// TIA Portal V18 export
FUNCTION "HeatingPLC_vIO" : Void   // FC11001, LAD
{ S7_Optimized_Access := 'FALSE' }
VERSION : 0.1
// stored: AutoNumber false, IsIECCheckEnabled false, SetENOAutomatically false, UDAEnableTagReadback false
BEGIN

REGION Network 1
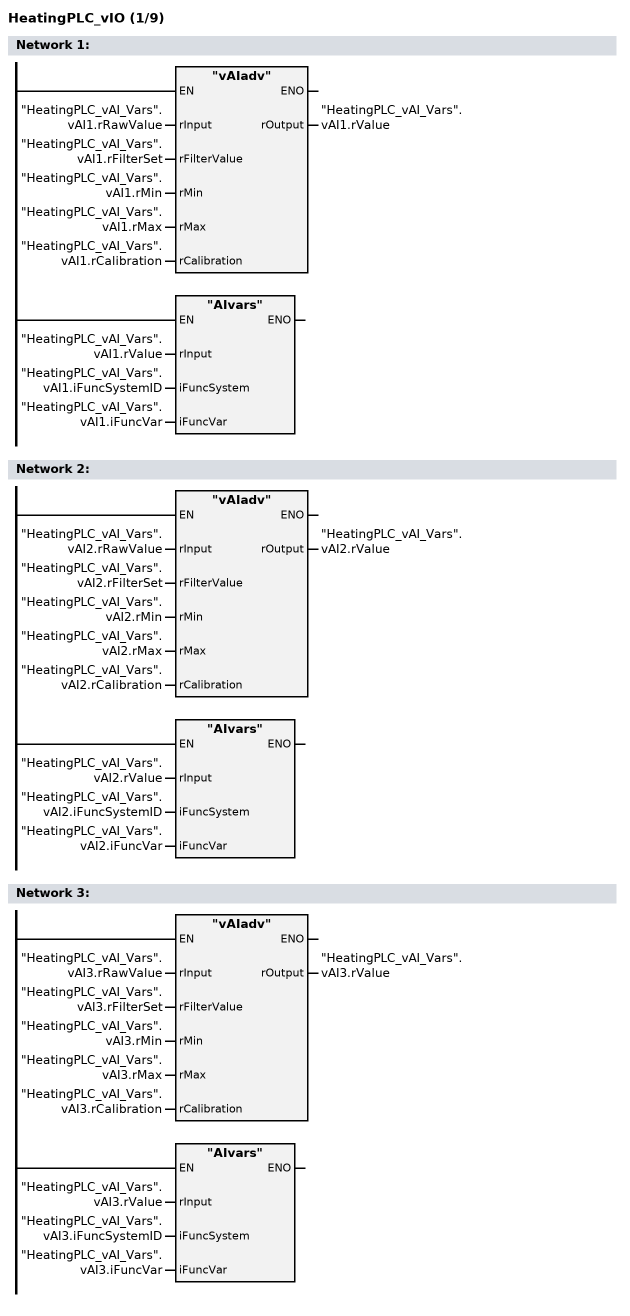
   RUNG wire#powerrail
      "vAIadv"(rInput := "HeatingPLC_vAI_Vars".vAI1.rRawValue, rFilterValue := "HeatingPLC_vAI_Vars".vAI1.rFilterSet, rMin := "HeatingPLC_vAI_Vars".vAI1.rMin, rMax := "HeatingPLC_vAI_Vars".vAI1.rMax, rCalibration := "HeatingPLC_vAI_Vars".vAI1.rCalibration, rOutput => "HeatingPLC_vAI_Vars".vAI1.rValue)
   END_RUNG
   RUNG wire#powerrail
      "AIvars"(rInput := "HeatingPLC_vAI_Vars".vAI1.rValue, iFuncSystem := "HeatingPLC_vAI_Vars".vAI1.iFuncSystemID, iFuncVar := "HeatingPLC_vAI_Vars".vAI1.iFuncVar)
   END_RUNG
   // the same network as SCL:
   "vAIadv"(rInput := "HeatingPLC_vAI_Vars".vAI1.rRawValue,
            rFilterValue := "HeatingPLC_vAI_Vars".vAI1.rFilterSet,
            rMin := "HeatingPLC_vAI_Vars".vAI1.rMin,
            rMax := "HeatingPLC_vAI_Vars".vAI1.rMax,
            rCalibration := "HeatingPLC_vAI_Vars".vAI1.rCalibration,
            rOutput => "HeatingPLC_vAI_Vars".vAI1.rValue);
   "AIvars"(rInput := "HeatingPLC_vAI_Vars".vAI1.rValue,
            iFuncSystem := "HeatingPLC_vAI_Vars".vAI1.iFuncSystemID,
            iFuncVar := "HeatingPLC_vAI_Vars".vAI1.iFuncVar);
END_REGION

REGION Network 2
   RUNG wire#powerrail
      "vAIadv"(rInput := "HeatingPLC_vAI_Vars".vAI2.rRawValue, rFilterValue := "HeatingPLC_vAI_Vars".vAI2.rFilterSet, rMin := "HeatingPLC_vAI_Vars".vAI2.rMin, rMax := "HeatingPLC_vAI_Vars".vAI2.rMax, rCalibration := "HeatingPLC_vAI_Vars".vAI2.rCalibration, rOutput => "HeatingPLC_vAI_Vars".vAI2.rValue)
   END_RUNG
   RUNG wire#powerrail
      "AIvars"(rInput := "HeatingPLC_vAI_Vars".vAI2.rValue, iFuncSystem := "HeatingPLC_vAI_Vars".vAI2.iFuncSystemID, iFuncVar := "HeatingPLC_vAI_Vars".vAI2.iFuncVar)
   END_RUNG
   // the same network as SCL:
   "vAIadv"(rInput := "HeatingPLC_vAI_Vars".vAI2.rRawValue,
            rFilterValue := "HeatingPLC_vAI_Vars".vAI2.rFilterSet,
            rMin := "HeatingPLC_vAI_Vars".vAI2.rMin,
            rMax := "HeatingPLC_vAI_Vars".vAI2.rMax,
            rCalibration := "HeatingPLC_vAI_Vars".vAI2.rCalibration,
            rOutput => "HeatingPLC_vAI_Vars".vAI2.rValue);
   "AIvars"(rInput := "HeatingPLC_vAI_Vars".vAI2.rValue,
            iFuncSystem := "HeatingPLC_vAI_Vars".vAI2.iFuncSystemID,
            iFuncVar := "HeatingPLC_vAI_Vars".vAI2.iFuncVar);
END_REGION

REGION Network 3
   RUNG wire#powerrail
      "vAIadv"(rInput := "HeatingPLC_vAI_Vars".vAI3.rRawValue, rFilterValue := "HeatingPLC_vAI_Vars".vAI3.rFilterSet, rMin := "HeatingPLC_vAI_Vars".vAI3.rMin, rMax := "HeatingPLC_vAI_Vars".vAI3.rMax, rCalibration := "HeatingPLC_vAI_Vars".vAI3.rCalibration, rOutput => "HeatingPLC_vAI_Vars".vAI3.rValue)
   END_RUNG
   RUNG wire#powerrail
      "AIvars"(rInput := "HeatingPLC_vAI_Vars".vAI3.rValue, iFuncSystem := "HeatingPLC_vAI_Vars".vAI3.iFuncSystemID, iFuncVar := "HeatingPLC_vAI_Vars".vAI3.iFuncVar)
   END_RUNG
   // the same network as SCL:
   "vAIadv"(rInput := "HeatingPLC_vAI_Vars".vAI3.rRawValue,
            rFilterValue := "HeatingPLC_vAI_Vars".vAI3.rFilterSet,
            rMin := "HeatingPLC_vAI_Vars".vAI3.rMin,
            rMax := "HeatingPLC_vAI_Vars".vAI3.rMax,
            rCalibration := "HeatingPLC_vAI_Vars".vAI3.rCalibration,
            rOutput => "HeatingPLC_vAI_Vars".vAI3.rValue);
   "AIvars"(rInput := "HeatingPLC_vAI_Vars".vAI3.rValue,
            iFuncSystem := "HeatingPLC_vAI_Vars".vAI3.iFuncSystemID,
            iFuncVar := "HeatingPLC_vAI_Vars".vAI3.iFuncVar);
END_REGION

REGION Network 4
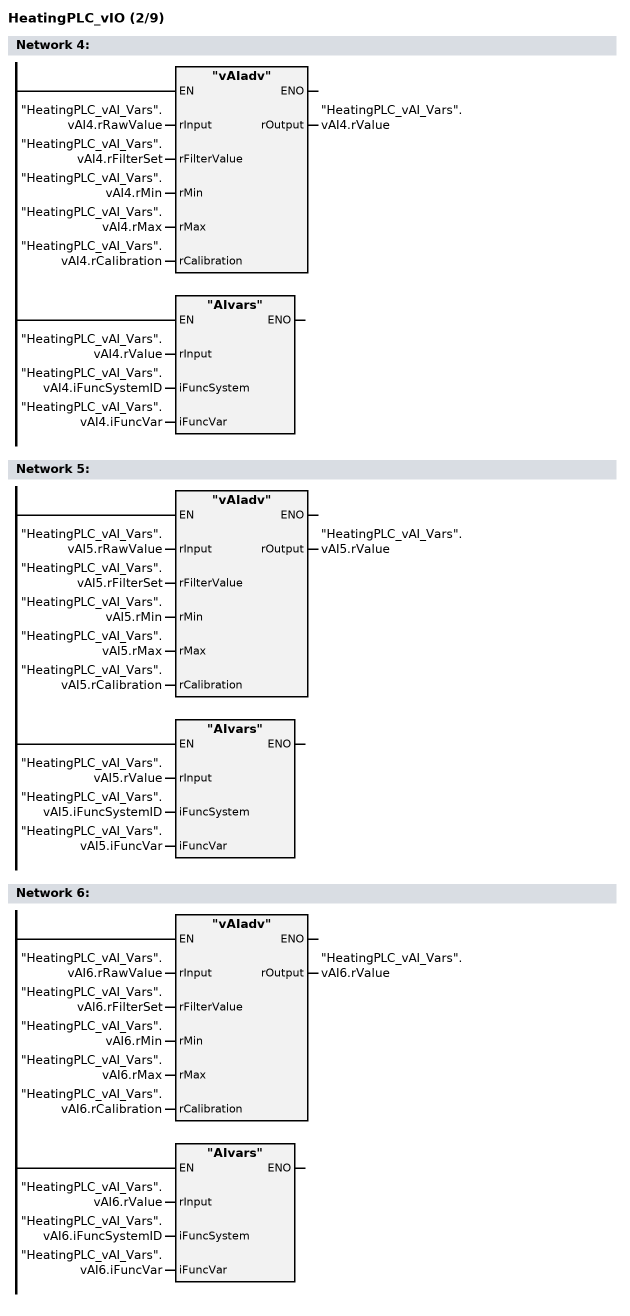
   RUNG wire#powerrail
      "vAIadv"(rInput := "HeatingPLC_vAI_Vars".vAI4.rRawValue, rFilterValue := "HeatingPLC_vAI_Vars".vAI4.rFilterSet, rMin := "HeatingPLC_vAI_Vars".vAI4.rMin, rMax := "HeatingPLC_vAI_Vars".vAI4.rMax, rCalibration := "HeatingPLC_vAI_Vars".vAI4.rCalibration, rOutput => "HeatingPLC_vAI_Vars".vAI4.rValue)
   END_RUNG
   RUNG wire#powerrail
      "AIvars"(rInput := "HeatingPLC_vAI_Vars".vAI4.rValue, iFuncSystem := "HeatingPLC_vAI_Vars".vAI4.iFuncSystemID, iFuncVar := "HeatingPLC_vAI_Vars".vAI4.iFuncVar)
   END_RUNG
   // the same network as SCL:
   "vAIadv"(rInput := "HeatingPLC_vAI_Vars".vAI4.rRawValue,
            rFilterValue := "HeatingPLC_vAI_Vars".vAI4.rFilterSet,
            rMin := "HeatingPLC_vAI_Vars".vAI4.rMin,
            rMax := "HeatingPLC_vAI_Vars".vAI4.rMax,
            rCalibration := "HeatingPLC_vAI_Vars".vAI4.rCalibration,
            rOutput => "HeatingPLC_vAI_Vars".vAI4.rValue);
   "AIvars"(rInput := "HeatingPLC_vAI_Vars".vAI4.rValue,
            iFuncSystem := "HeatingPLC_vAI_Vars".vAI4.iFuncSystemID,
            iFuncVar := "HeatingPLC_vAI_Vars".vAI4.iFuncVar);
END_REGION

REGION Network 5
   RUNG wire#powerrail
      "vAIadv"(rInput := "HeatingPLC_vAI_Vars".vAI5.rRawValue, rFilterValue := "HeatingPLC_vAI_Vars".vAI5.rFilterSet, rMin := "HeatingPLC_vAI_Vars".vAI5.rMin, rMax := "HeatingPLC_vAI_Vars".vAI5.rMax, rCalibration := "HeatingPLC_vAI_Vars".vAI5.rCalibration, rOutput => "HeatingPLC_vAI_Vars".vAI5.rValue)
   END_RUNG
   RUNG wire#powerrail
      "AIvars"(rInput := "HeatingPLC_vAI_Vars".vAI5.rValue, iFuncSystem := "HeatingPLC_vAI_Vars".vAI5.iFuncSystemID, iFuncVar := "HeatingPLC_vAI_Vars".vAI5.iFuncVar)
   END_RUNG
   // the same network as SCL:
   "vAIadv"(rInput := "HeatingPLC_vAI_Vars".vAI5.rRawValue,
            rFilterValue := "HeatingPLC_vAI_Vars".vAI5.rFilterSet,
            rMin := "HeatingPLC_vAI_Vars".vAI5.rMin,
            rMax := "HeatingPLC_vAI_Vars".vAI5.rMax,
            rCalibration := "HeatingPLC_vAI_Vars".vAI5.rCalibration,
            rOutput => "HeatingPLC_vAI_Vars".vAI5.rValue);
   "AIvars"(rInput := "HeatingPLC_vAI_Vars".vAI5.rValue,
            iFuncSystem := "HeatingPLC_vAI_Vars".vAI5.iFuncSystemID,
            iFuncVar := "HeatingPLC_vAI_Vars".vAI5.iFuncVar);
END_REGION

REGION Network 6
   RUNG wire#powerrail
      "vAIadv"(rInput := "HeatingPLC_vAI_Vars".vAI6.rRawValue, rFilterValue := "HeatingPLC_vAI_Vars".vAI6.rFilterSet, rMin := "HeatingPLC_vAI_Vars".vAI6.rMin, rMax := "HeatingPLC_vAI_Vars".vAI6.rMax, rCalibration := "HeatingPLC_vAI_Vars".vAI6.rCalibration, rOutput => "HeatingPLC_vAI_Vars".vAI6.rValue)
   END_RUNG
   RUNG wire#powerrail
      "AIvars"(rInput := "HeatingPLC_vAI_Vars".vAI6.rValue, iFuncSystem := "HeatingPLC_vAI_Vars".vAI6.iFuncSystemID, iFuncVar := "HeatingPLC_vAI_Vars".vAI6.iFuncVar)
   END_RUNG
   // the same network as SCL:
   "vAIadv"(rInput := "HeatingPLC_vAI_Vars".vAI6.rRawValue,
            rFilterValue := "HeatingPLC_vAI_Vars".vAI6.rFilterSet,
            rMin := "HeatingPLC_vAI_Vars".vAI6.rMin,
            rMax := "HeatingPLC_vAI_Vars".vAI6.rMax,
            rCalibration := "HeatingPLC_vAI_Vars".vAI6.rCalibration,
            rOutput => "HeatingPLC_vAI_Vars".vAI6.rValue);
   "AIvars"(rInput := "HeatingPLC_vAI_Vars".vAI6.rValue,
            iFuncSystem := "HeatingPLC_vAI_Vars".vAI6.iFuncSystemID,
            iFuncVar := "HeatingPLC_vAI_Vars".vAI6.iFuncVar);
END_REGION

REGION Network 7
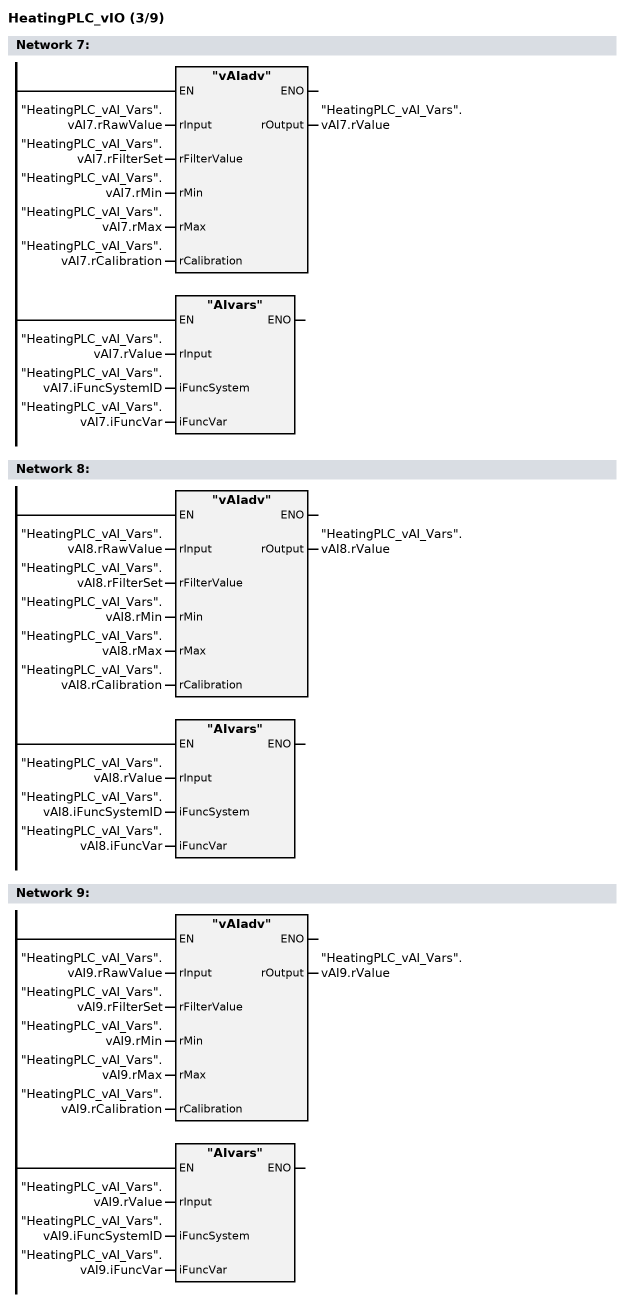
   RUNG wire#powerrail
      "vAIadv"(rInput := "HeatingPLC_vAI_Vars".vAI7.rRawValue, rFilterValue := "HeatingPLC_vAI_Vars".vAI7.rFilterSet, rMin := "HeatingPLC_vAI_Vars".vAI7.rMin, rMax := "HeatingPLC_vAI_Vars".vAI7.rMax, rCalibration := "HeatingPLC_vAI_Vars".vAI7.rCalibration, rOutput => "HeatingPLC_vAI_Vars".vAI7.rValue)
   END_RUNG
   RUNG wire#powerrail
      "AIvars"(rInput := "HeatingPLC_vAI_Vars".vAI7.rValue, iFuncSystem := "HeatingPLC_vAI_Vars".vAI7.iFuncSystemID, iFuncVar := "HeatingPLC_vAI_Vars".vAI7.iFuncVar)
   END_RUNG
   // the same network as SCL:
   "vAIadv"(rInput := "HeatingPLC_vAI_Vars".vAI7.rRawValue,
            rFilterValue := "HeatingPLC_vAI_Vars".vAI7.rFilterSet,
            rMin := "HeatingPLC_vAI_Vars".vAI7.rMin,
            rMax := "HeatingPLC_vAI_Vars".vAI7.rMax,
            rCalibration := "HeatingPLC_vAI_Vars".vAI7.rCalibration,
            rOutput => "HeatingPLC_vAI_Vars".vAI7.rValue);
   "AIvars"(rInput := "HeatingPLC_vAI_Vars".vAI7.rValue,
            iFuncSystem := "HeatingPLC_vAI_Vars".vAI7.iFuncSystemID,
            iFuncVar := "HeatingPLC_vAI_Vars".vAI7.iFuncVar);
END_REGION

REGION Network 8
   RUNG wire#powerrail
      "vAIadv"(rInput := "HeatingPLC_vAI_Vars".vAI8.rRawValue, rFilterValue := "HeatingPLC_vAI_Vars".vAI8.rFilterSet, rMin := "HeatingPLC_vAI_Vars".vAI8.rMin, rMax := "HeatingPLC_vAI_Vars".vAI8.rMax, rCalibration := "HeatingPLC_vAI_Vars".vAI8.rCalibration, rOutput => "HeatingPLC_vAI_Vars".vAI8.rValue)
   END_RUNG
   RUNG wire#powerrail
      "AIvars"(rInput := "HeatingPLC_vAI_Vars".vAI8.rValue, iFuncSystem := "HeatingPLC_vAI_Vars".vAI8.iFuncSystemID, iFuncVar := "HeatingPLC_vAI_Vars".vAI8.iFuncVar)
   END_RUNG
   // the same network as SCL:
   "vAIadv"(rInput := "HeatingPLC_vAI_Vars".vAI8.rRawValue,
            rFilterValue := "HeatingPLC_vAI_Vars".vAI8.rFilterSet,
            rMin := "HeatingPLC_vAI_Vars".vAI8.rMin,
            rMax := "HeatingPLC_vAI_Vars".vAI8.rMax,
            rCalibration := "HeatingPLC_vAI_Vars".vAI8.rCalibration,
            rOutput => "HeatingPLC_vAI_Vars".vAI8.rValue);
   "AIvars"(rInput := "HeatingPLC_vAI_Vars".vAI8.rValue,
            iFuncSystem := "HeatingPLC_vAI_Vars".vAI8.iFuncSystemID,
            iFuncVar := "HeatingPLC_vAI_Vars".vAI8.iFuncVar);
END_REGION

REGION Network 9
   RUNG wire#powerrail
      "vAIadv"(rInput := "HeatingPLC_vAI_Vars".vAI9.rRawValue, rFilterValue := "HeatingPLC_vAI_Vars".vAI9.rFilterSet, rMin := "HeatingPLC_vAI_Vars".vAI9.rMin, rMax := "HeatingPLC_vAI_Vars".vAI9.rMax, rCalibration := "HeatingPLC_vAI_Vars".vAI9.rCalibration, rOutput => "HeatingPLC_vAI_Vars".vAI9.rValue)
   END_RUNG
   RUNG wire#powerrail
      "AIvars"(rInput := "HeatingPLC_vAI_Vars".vAI9.rValue, iFuncSystem := "HeatingPLC_vAI_Vars".vAI9.iFuncSystemID, iFuncVar := "HeatingPLC_vAI_Vars".vAI9.iFuncVar)
   END_RUNG
   // the same network as SCL:
   "vAIadv"(rInput := "HeatingPLC_vAI_Vars".vAI9.rRawValue,
            rFilterValue := "HeatingPLC_vAI_Vars".vAI9.rFilterSet,
            rMin := "HeatingPLC_vAI_Vars".vAI9.rMin,
            rMax := "HeatingPLC_vAI_Vars".vAI9.rMax,
            rCalibration := "HeatingPLC_vAI_Vars".vAI9.rCalibration,
            rOutput => "HeatingPLC_vAI_Vars".vAI9.rValue);
   "AIvars"(rInput := "HeatingPLC_vAI_Vars".vAI9.rValue,
            iFuncSystem := "HeatingPLC_vAI_Vars".vAI9.iFuncSystemID,
            iFuncVar := "HeatingPLC_vAI_Vars".vAI9.iFuncVar);
END_REGION

REGION Network 10
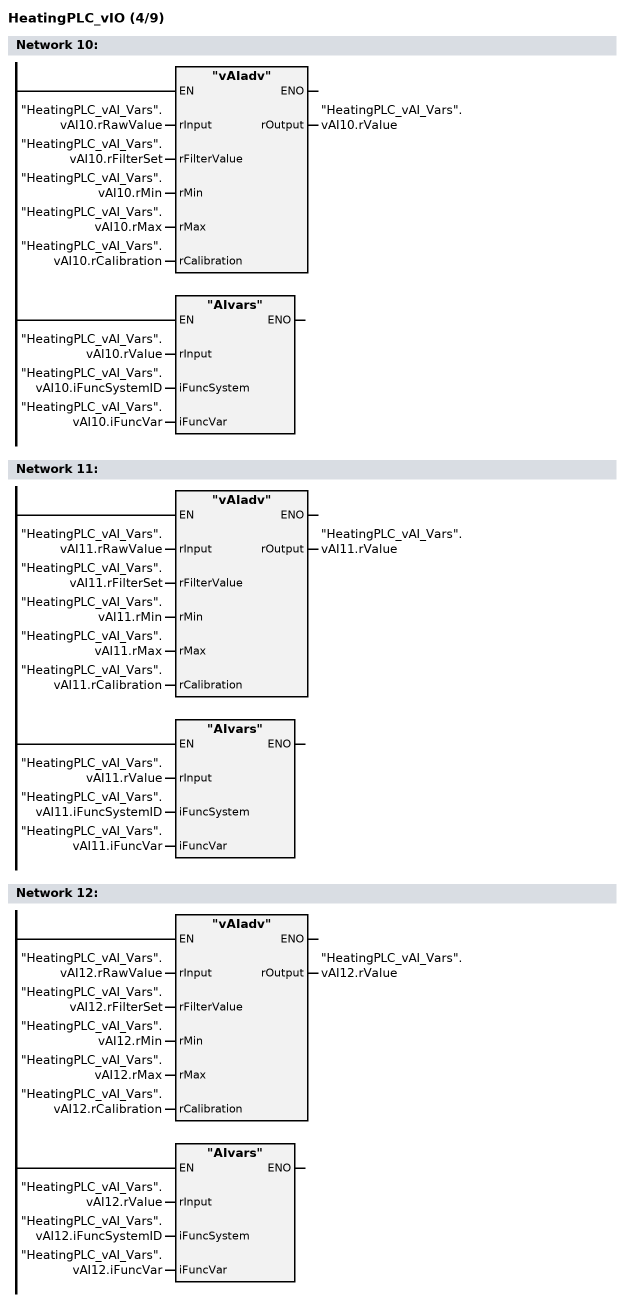
   RUNG wire#powerrail
      "vAIadv"(rInput := "HeatingPLC_vAI_Vars".vAI10.rRawValue, rFilterValue := "HeatingPLC_vAI_Vars".vAI10.rFilterSet, rMin := "HeatingPLC_vAI_Vars".vAI10.rMin, rMax := "HeatingPLC_vAI_Vars".vAI10.rMax, rCalibration := "HeatingPLC_vAI_Vars".vAI10.rCalibration, rOutput => "HeatingPLC_vAI_Vars".vAI10.rValue)
   END_RUNG
   RUNG wire#powerrail
      "AIvars"(rInput := "HeatingPLC_vAI_Vars".vAI10.rValue, iFuncSystem := "HeatingPLC_vAI_Vars".vAI10.iFuncSystemID, iFuncVar := "HeatingPLC_vAI_Vars".vAI10.iFuncVar)
   END_RUNG
   // the same network as SCL:
   "vAIadv"(rInput := "HeatingPLC_vAI_Vars".vAI10.rRawValue,
            rFilterValue := "HeatingPLC_vAI_Vars".vAI10.rFilterSet,
            rMin := "HeatingPLC_vAI_Vars".vAI10.rMin,
            rMax := "HeatingPLC_vAI_Vars".vAI10.rMax,
            rCalibration := "HeatingPLC_vAI_Vars".vAI10.rCalibration,
            rOutput => "HeatingPLC_vAI_Vars".vAI10.rValue);
   "AIvars"(rInput := "HeatingPLC_vAI_Vars".vAI10.rValue,
            iFuncSystem := "HeatingPLC_vAI_Vars".vAI10.iFuncSystemID,
            iFuncVar := "HeatingPLC_vAI_Vars".vAI10.iFuncVar);
END_REGION

REGION Network 11
   RUNG wire#powerrail
      "vAIadv"(rInput := "HeatingPLC_vAI_Vars".vAI11.rRawValue, rFilterValue := "HeatingPLC_vAI_Vars".vAI11.rFilterSet, rMin := "HeatingPLC_vAI_Vars".vAI11.rMin, rMax := "HeatingPLC_vAI_Vars".vAI11.rMax, rCalibration := "HeatingPLC_vAI_Vars".vAI11.rCalibration, rOutput => "HeatingPLC_vAI_Vars".vAI11.rValue)
   END_RUNG
   RUNG wire#powerrail
      "AIvars"(rInput := "HeatingPLC_vAI_Vars".vAI11.rValue, iFuncSystem := "HeatingPLC_vAI_Vars".vAI11.iFuncSystemID, iFuncVar := "HeatingPLC_vAI_Vars".vAI11.iFuncVar)
   END_RUNG
   // the same network as SCL:
   "vAIadv"(rInput := "HeatingPLC_vAI_Vars".vAI11.rRawValue,
            rFilterValue := "HeatingPLC_vAI_Vars".vAI11.rFilterSet,
            rMin := "HeatingPLC_vAI_Vars".vAI11.rMin,
            rMax := "HeatingPLC_vAI_Vars".vAI11.rMax,
            rCalibration := "HeatingPLC_vAI_Vars".vAI11.rCalibration,
            rOutput => "HeatingPLC_vAI_Vars".vAI11.rValue);
   "AIvars"(rInput := "HeatingPLC_vAI_Vars".vAI11.rValue,
            iFuncSystem := "HeatingPLC_vAI_Vars".vAI11.iFuncSystemID,
            iFuncVar := "HeatingPLC_vAI_Vars".vAI11.iFuncVar);
END_REGION

REGION Network 12
   RUNG wire#powerrail
      "vAIadv"(rInput := "HeatingPLC_vAI_Vars".vAI12.rRawValue, rFilterValue := "HeatingPLC_vAI_Vars".vAI12.rFilterSet, rMin := "HeatingPLC_vAI_Vars".vAI12.rMin, rMax := "HeatingPLC_vAI_Vars".vAI12.rMax, rCalibration := "HeatingPLC_vAI_Vars".vAI12.rCalibration, rOutput => "HeatingPLC_vAI_Vars".vAI12.rValue)
   END_RUNG
   RUNG wire#powerrail
      "AIvars"(rInput := "HeatingPLC_vAI_Vars".vAI12.rValue, iFuncSystem := "HeatingPLC_vAI_Vars".vAI12.iFuncSystemID, iFuncVar := "HeatingPLC_vAI_Vars".vAI12.iFuncVar)
   END_RUNG
   // the same network as SCL:
   "vAIadv"(rInput := "HeatingPLC_vAI_Vars".vAI12.rRawValue,
            rFilterValue := "HeatingPLC_vAI_Vars".vAI12.rFilterSet,
            rMin := "HeatingPLC_vAI_Vars".vAI12.rMin,
            rMax := "HeatingPLC_vAI_Vars".vAI12.rMax,
            rCalibration := "HeatingPLC_vAI_Vars".vAI12.rCalibration,
            rOutput => "HeatingPLC_vAI_Vars".vAI12.rValue);
   "AIvars"(rInput := "HeatingPLC_vAI_Vars".vAI12.rValue,
            iFuncSystem := "HeatingPLC_vAI_Vars".vAI12.iFuncSystemID,
            iFuncVar := "HeatingPLC_vAI_Vars".vAI12.iFuncVar);
END_REGION

REGION Network 13
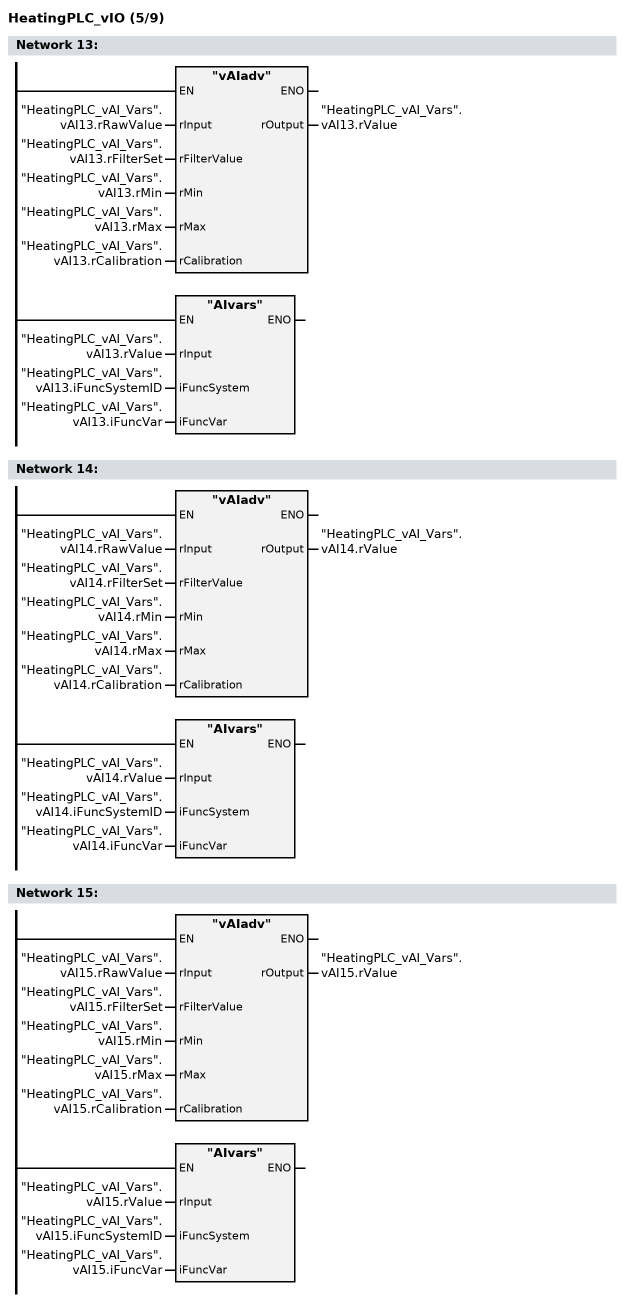
   RUNG wire#powerrail
      "vAIadv"(rInput := "HeatingPLC_vAI_Vars".vAI13.rRawValue, rFilterValue := "HeatingPLC_vAI_Vars".vAI13.rFilterSet, rMin := "HeatingPLC_vAI_Vars".vAI13.rMin, rMax := "HeatingPLC_vAI_Vars".vAI13.rMax, rCalibration := "HeatingPLC_vAI_Vars".vAI13.rCalibration, rOutput => "HeatingPLC_vAI_Vars".vAI13.rValue)
   END_RUNG
   RUNG wire#powerrail
      "AIvars"(rInput := "HeatingPLC_vAI_Vars".vAI13.rValue, iFuncSystem := "HeatingPLC_vAI_Vars".vAI13.iFuncSystemID, iFuncVar := "HeatingPLC_vAI_Vars".vAI13.iFuncVar)
   END_RUNG
   // the same network as SCL:
   "vAIadv"(rInput := "HeatingPLC_vAI_Vars".vAI13.rRawValue,
            rFilterValue := "HeatingPLC_vAI_Vars".vAI13.rFilterSet,
            rMin := "HeatingPLC_vAI_Vars".vAI13.rMin,
            rMax := "HeatingPLC_vAI_Vars".vAI13.rMax,
            rCalibration := "HeatingPLC_vAI_Vars".vAI13.rCalibration,
            rOutput => "HeatingPLC_vAI_Vars".vAI13.rValue);
   "AIvars"(rInput := "HeatingPLC_vAI_Vars".vAI13.rValue,
            iFuncSystem := "HeatingPLC_vAI_Vars".vAI13.iFuncSystemID,
            iFuncVar := "HeatingPLC_vAI_Vars".vAI13.iFuncVar);
END_REGION

REGION Network 14
   RUNG wire#powerrail
      "vAIadv"(rInput := "HeatingPLC_vAI_Vars".vAI14.rRawValue, rFilterValue := "HeatingPLC_vAI_Vars".vAI14.rFilterSet, rMin := "HeatingPLC_vAI_Vars".vAI14.rMin, rMax := "HeatingPLC_vAI_Vars".vAI14.rMax, rCalibration := "HeatingPLC_vAI_Vars".vAI14.rCalibration, rOutput => "HeatingPLC_vAI_Vars".vAI14.rValue)
   END_RUNG
   RUNG wire#powerrail
      "AIvars"(rInput := "HeatingPLC_vAI_Vars".vAI14.rValue, iFuncSystem := "HeatingPLC_vAI_Vars".vAI14.iFuncSystemID, iFuncVar := "HeatingPLC_vAI_Vars".vAI14.iFuncVar)
   END_RUNG
   // the same network as SCL:
   "vAIadv"(rInput := "HeatingPLC_vAI_Vars".vAI14.rRawValue,
            rFilterValue := "HeatingPLC_vAI_Vars".vAI14.rFilterSet,
            rMin := "HeatingPLC_vAI_Vars".vAI14.rMin,
            rMax := "HeatingPLC_vAI_Vars".vAI14.rMax,
            rCalibration := "HeatingPLC_vAI_Vars".vAI14.rCalibration,
            rOutput => "HeatingPLC_vAI_Vars".vAI14.rValue);
   "AIvars"(rInput := "HeatingPLC_vAI_Vars".vAI14.rValue,
            iFuncSystem := "HeatingPLC_vAI_Vars".vAI14.iFuncSystemID,
            iFuncVar := "HeatingPLC_vAI_Vars".vAI14.iFuncVar);
END_REGION

REGION Network 15
   RUNG wire#powerrail
      "vAIadv"(rInput := "HeatingPLC_vAI_Vars".vAI15.rRawValue, rFilterValue := "HeatingPLC_vAI_Vars".vAI15.rFilterSet, rMin := "HeatingPLC_vAI_Vars".vAI15.rMin, rMax := "HeatingPLC_vAI_Vars".vAI15.rMax, rCalibration := "HeatingPLC_vAI_Vars".vAI15.rCalibration, rOutput => "HeatingPLC_vAI_Vars".vAI15.rValue)
   END_RUNG
   RUNG wire#powerrail
      "AIvars"(rInput := "HeatingPLC_vAI_Vars".vAI15.rValue, iFuncSystem := "HeatingPLC_vAI_Vars".vAI15.iFuncSystemID, iFuncVar := "HeatingPLC_vAI_Vars".vAI15.iFuncVar)
   END_RUNG
   // the same network as SCL:
   "vAIadv"(rInput := "HeatingPLC_vAI_Vars".vAI15.rRawValue,
            rFilterValue := "HeatingPLC_vAI_Vars".vAI15.rFilterSet,
            rMin := "HeatingPLC_vAI_Vars".vAI15.rMin,
            rMax := "HeatingPLC_vAI_Vars".vAI15.rMax,
            rCalibration := "HeatingPLC_vAI_Vars".vAI15.rCalibration,
            rOutput => "HeatingPLC_vAI_Vars".vAI15.rValue);
   "AIvars"(rInput := "HeatingPLC_vAI_Vars".vAI15.rValue,
            iFuncSystem := "HeatingPLC_vAI_Vars".vAI15.iFuncSystemID,
            iFuncVar := "HeatingPLC_vAI_Vars".vAI15.iFuncVar);
END_REGION

REGION Network 16
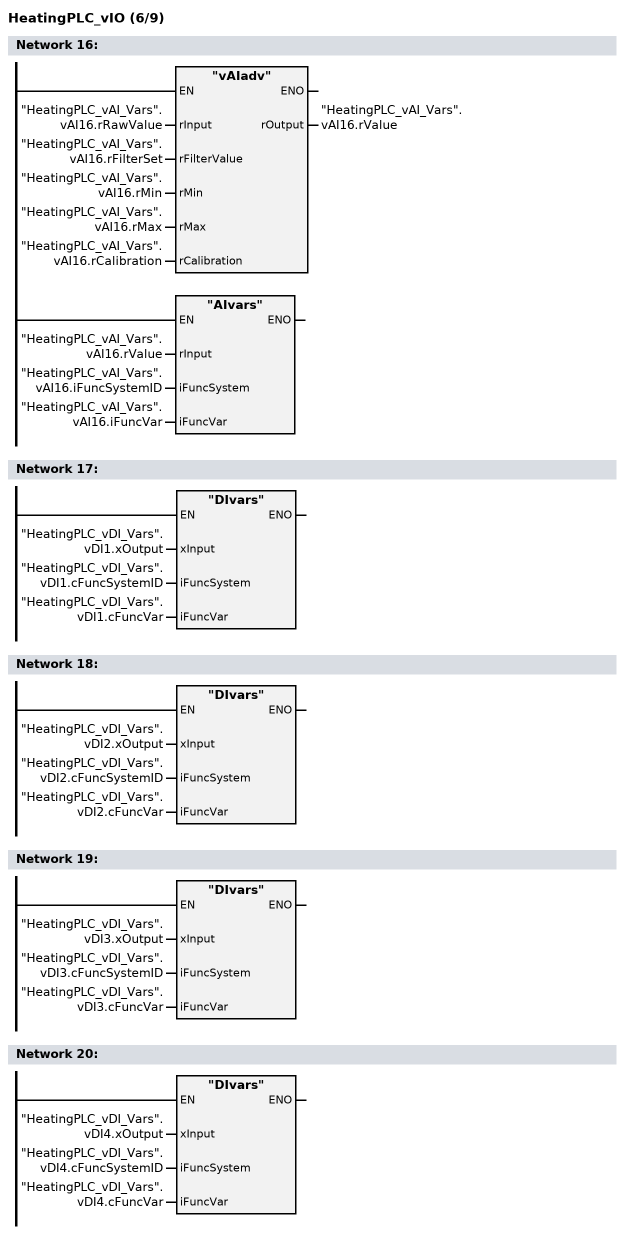
   RUNG wire#powerrail
      "vAIadv"(rInput := "HeatingPLC_vAI_Vars".vAI16.rRawValue, rFilterValue := "HeatingPLC_vAI_Vars".vAI16.rFilterSet, rMin := "HeatingPLC_vAI_Vars".vAI16.rMin, rMax := "HeatingPLC_vAI_Vars".vAI16.rMax, rCalibration := "HeatingPLC_vAI_Vars".vAI16.rCalibration, rOutput => "HeatingPLC_vAI_Vars".vAI16.rValue)
   END_RUNG
   RUNG wire#powerrail
      "AIvars"(rInput := "HeatingPLC_vAI_Vars".vAI16.rValue, iFuncSystem := "HeatingPLC_vAI_Vars".vAI16.iFuncSystemID, iFuncVar := "HeatingPLC_vAI_Vars".vAI16.iFuncVar)
   END_RUNG
   // the same network as SCL:
   "vAIadv"(rInput := "HeatingPLC_vAI_Vars".vAI16.rRawValue,
            rFilterValue := "HeatingPLC_vAI_Vars".vAI16.rFilterSet,
            rMin := "HeatingPLC_vAI_Vars".vAI16.rMin,
            rMax := "HeatingPLC_vAI_Vars".vAI16.rMax,
            rCalibration := "HeatingPLC_vAI_Vars".vAI16.rCalibration,
            rOutput => "HeatingPLC_vAI_Vars".vAI16.rValue);
   "AIvars"(rInput := "HeatingPLC_vAI_Vars".vAI16.rValue,
            iFuncSystem := "HeatingPLC_vAI_Vars".vAI16.iFuncSystemID,
            iFuncVar := "HeatingPLC_vAI_Vars".vAI16.iFuncVar);
END_REGION

REGION Network 17
   RUNG wire#powerrail
      "DIvars"(xInput := "HeatingPLC_vDI_Vars".vDI1.xOutput, iFuncSystem := "HeatingPLC_vDI_Vars".vDI1.cFuncSystemID, iFuncVar := "HeatingPLC_vDI_Vars".vDI1.cFuncVar)
   END_RUNG
   // the same network as SCL:
   "DIvars"(xInput := "HeatingPLC_vDI_Vars".vDI1.xOutput,
            iFuncSystem := "HeatingPLC_vDI_Vars".vDI1.cFuncSystemID,
            iFuncVar := "HeatingPLC_vDI_Vars".vDI1.cFuncVar);
END_REGION

REGION Network 18
   RUNG wire#powerrail
      "DIvars"(xInput := "HeatingPLC_vDI_Vars".vDI2.xOutput, iFuncSystem := "HeatingPLC_vDI_Vars".vDI2.cFuncSystemID, iFuncVar := "HeatingPLC_vDI_Vars".vDI2.cFuncVar)
   END_RUNG
   // the same network as SCL:
   "DIvars"(xInput := "HeatingPLC_vDI_Vars".vDI2.xOutput,
            iFuncSystem := "HeatingPLC_vDI_Vars".vDI2.cFuncSystemID,
            iFuncVar := "HeatingPLC_vDI_Vars".vDI2.cFuncVar);
END_REGION

REGION Network 19
   RUNG wire#powerrail
      "DIvars"(xInput := "HeatingPLC_vDI_Vars".vDI3.xOutput, iFuncSystem := "HeatingPLC_vDI_Vars".vDI3.cFuncSystemID, iFuncVar := "HeatingPLC_vDI_Vars".vDI3.cFuncVar)
   END_RUNG
   // the same network as SCL:
   "DIvars"(xInput := "HeatingPLC_vDI_Vars".vDI3.xOutput,
            iFuncSystem := "HeatingPLC_vDI_Vars".vDI3.cFuncSystemID,
            iFuncVar := "HeatingPLC_vDI_Vars".vDI3.cFuncVar);
END_REGION

REGION Network 20
   RUNG wire#powerrail
      "DIvars"(xInput := "HeatingPLC_vDI_Vars".vDI4.xOutput, iFuncSystem := "HeatingPLC_vDI_Vars".vDI4.cFuncSystemID, iFuncVar := "HeatingPLC_vDI_Vars".vDI4.cFuncVar)
   END_RUNG
   // the same network as SCL:
   "DIvars"(xInput := "HeatingPLC_vDI_Vars".vDI4.xOutput,
            iFuncSystem := "HeatingPLC_vDI_Vars".vDI4.cFuncSystemID,
            iFuncVar := "HeatingPLC_vDI_Vars".vDI4.cFuncVar);
END_REGION

REGION Network 21
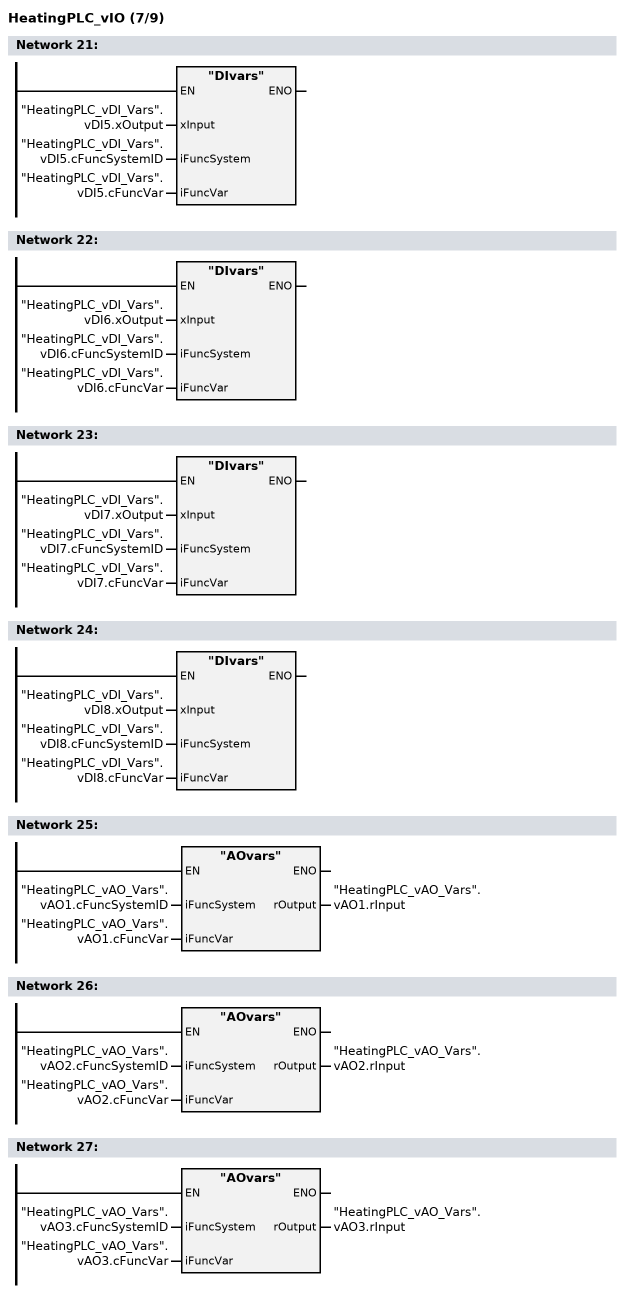
   RUNG wire#powerrail
      "DIvars"(xInput := "HeatingPLC_vDI_Vars".vDI5.xOutput, iFuncSystem := "HeatingPLC_vDI_Vars".vDI5.cFuncSystemID, iFuncVar := "HeatingPLC_vDI_Vars".vDI5.cFuncVar)
   END_RUNG
   // the same network as SCL:
   "DIvars"(xInput := "HeatingPLC_vDI_Vars".vDI5.xOutput,
            iFuncSystem := "HeatingPLC_vDI_Vars".vDI5.cFuncSystemID,
            iFuncVar := "HeatingPLC_vDI_Vars".vDI5.cFuncVar);
END_REGION

REGION Network 22
   RUNG wire#powerrail
      "DIvars"(xInput := "HeatingPLC_vDI_Vars".vDI6.xOutput, iFuncSystem := "HeatingPLC_vDI_Vars".vDI6.cFuncSystemID, iFuncVar := "HeatingPLC_vDI_Vars".vDI6.cFuncVar)
   END_RUNG
   // the same network as SCL:
   "DIvars"(xInput := "HeatingPLC_vDI_Vars".vDI6.xOutput,
            iFuncSystem := "HeatingPLC_vDI_Vars".vDI6.cFuncSystemID,
            iFuncVar := "HeatingPLC_vDI_Vars".vDI6.cFuncVar);
END_REGION

REGION Network 23
   RUNG wire#powerrail
      "DIvars"(xInput := "HeatingPLC_vDI_Vars".vDI7.xOutput, iFuncSystem := "HeatingPLC_vDI_Vars".vDI7.cFuncSystemID, iFuncVar := "HeatingPLC_vDI_Vars".vDI7.cFuncVar)
   END_RUNG
   // the same network as SCL:
   "DIvars"(xInput := "HeatingPLC_vDI_Vars".vDI7.xOutput,
            iFuncSystem := "HeatingPLC_vDI_Vars".vDI7.cFuncSystemID,
            iFuncVar := "HeatingPLC_vDI_Vars".vDI7.cFuncVar);
END_REGION

REGION Network 24
   RUNG wire#powerrail
      "DIvars"(xInput := "HeatingPLC_vDI_Vars".vDI8.xOutput, iFuncSystem := "HeatingPLC_vDI_Vars".vDI8.cFuncSystemID, iFuncVar := "HeatingPLC_vDI_Vars".vDI8.cFuncVar)
   END_RUNG
   // the same network as SCL:
   "DIvars"(xInput := "HeatingPLC_vDI_Vars".vDI8.xOutput,
            iFuncSystem := "HeatingPLC_vDI_Vars".vDI8.cFuncSystemID,
            iFuncVar := "HeatingPLC_vDI_Vars".vDI8.cFuncVar);
END_REGION

REGION Network 25
   RUNG wire#powerrail
      "AOvars"(iFuncSystem := "HeatingPLC_vAO_Vars".vAO1.cFuncSystemID, iFuncVar := "HeatingPLC_vAO_Vars".vAO1.cFuncVar, rOutput => "HeatingPLC_vAO_Vars".vAO1.rInput)
   END_RUNG
   // the same network as SCL:
   "AOvars"(iFuncSystem := "HeatingPLC_vAO_Vars".vAO1.cFuncSystemID,
            iFuncVar := "HeatingPLC_vAO_Vars".vAO1.cFuncVar,
            rOutput => "HeatingPLC_vAO_Vars".vAO1.rInput);
END_REGION

REGION Network 26
   RUNG wire#powerrail
      "AOvars"(iFuncSystem := "HeatingPLC_vAO_Vars".vAO2.cFuncSystemID, iFuncVar := "HeatingPLC_vAO_Vars".vAO2.cFuncVar, rOutput => "HeatingPLC_vAO_Vars".vAO2.rInput)
   END_RUNG
   // the same network as SCL:
   "AOvars"(iFuncSystem := "HeatingPLC_vAO_Vars".vAO2.cFuncSystemID,
            iFuncVar := "HeatingPLC_vAO_Vars".vAO2.cFuncVar,
            rOutput => "HeatingPLC_vAO_Vars".vAO2.rInput);
END_REGION

REGION Network 27
   RUNG wire#powerrail
      "AOvars"(iFuncSystem := "HeatingPLC_vAO_Vars".vAO3.cFuncSystemID, iFuncVar := "HeatingPLC_vAO_Vars".vAO3.cFuncVar, rOutput => "HeatingPLC_vAO_Vars".vAO3.rInput)
   END_RUNG
   // the same network as SCL:
   "AOvars"(iFuncSystem := "HeatingPLC_vAO_Vars".vAO3.cFuncSystemID,
            iFuncVar := "HeatingPLC_vAO_Vars".vAO3.cFuncVar,
            rOutput => "HeatingPLC_vAO_Vars".vAO3.rInput);
END_REGION

REGION Network 28
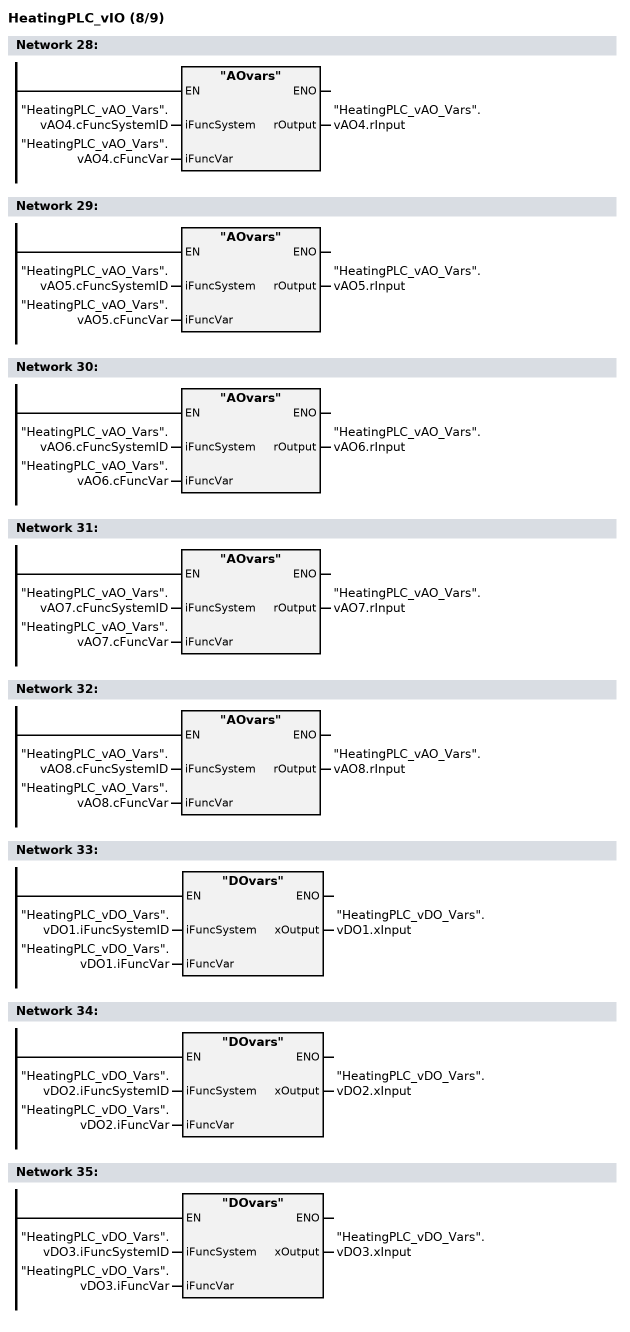
   RUNG wire#powerrail
      "AOvars"(iFuncSystem := "HeatingPLC_vAO_Vars".vAO4.cFuncSystemID, iFuncVar := "HeatingPLC_vAO_Vars".vAO4.cFuncVar, rOutput => "HeatingPLC_vAO_Vars".vAO4.rInput)
   END_RUNG
   // the same network as SCL:
   "AOvars"(iFuncSystem := "HeatingPLC_vAO_Vars".vAO4.cFuncSystemID,
            iFuncVar := "HeatingPLC_vAO_Vars".vAO4.cFuncVar,
            rOutput => "HeatingPLC_vAO_Vars".vAO4.rInput);
END_REGION

REGION Network 29
   RUNG wire#powerrail
      "AOvars"(iFuncSystem := "HeatingPLC_vAO_Vars".vAO5.cFuncSystemID, iFuncVar := "HeatingPLC_vAO_Vars".vAO5.cFuncVar, rOutput => "HeatingPLC_vAO_Vars".vAO5.rInput)
   END_RUNG
   // the same network as SCL:
   "AOvars"(iFuncSystem := "HeatingPLC_vAO_Vars".vAO5.cFuncSystemID,
            iFuncVar := "HeatingPLC_vAO_Vars".vAO5.cFuncVar,
            rOutput => "HeatingPLC_vAO_Vars".vAO5.rInput);
END_REGION

REGION Network 30
   RUNG wire#powerrail
      "AOvars"(iFuncSystem := "HeatingPLC_vAO_Vars".vAO6.cFuncSystemID, iFuncVar := "HeatingPLC_vAO_Vars".vAO6.cFuncVar, rOutput => "HeatingPLC_vAO_Vars".vAO6.rInput)
   END_RUNG
   // the same network as SCL:
   "AOvars"(iFuncSystem := "HeatingPLC_vAO_Vars".vAO6.cFuncSystemID,
            iFuncVar := "HeatingPLC_vAO_Vars".vAO6.cFuncVar,
            rOutput => "HeatingPLC_vAO_Vars".vAO6.rInput);
END_REGION

REGION Network 31
   RUNG wire#powerrail
      "AOvars"(iFuncSystem := "HeatingPLC_vAO_Vars".vAO7.cFuncSystemID, iFuncVar := "HeatingPLC_vAO_Vars".vAO7.cFuncVar, rOutput => "HeatingPLC_vAO_Vars".vAO7.rInput)
   END_RUNG
   // the same network as SCL:
   "AOvars"(iFuncSystem := "HeatingPLC_vAO_Vars".vAO7.cFuncSystemID,
            iFuncVar := "HeatingPLC_vAO_Vars".vAO7.cFuncVar,
            rOutput => "HeatingPLC_vAO_Vars".vAO7.rInput);
END_REGION

REGION Network 32
   RUNG wire#powerrail
      "AOvars"(iFuncSystem := "HeatingPLC_vAO_Vars".vAO8.cFuncSystemID, iFuncVar := "HeatingPLC_vAO_Vars".vAO8.cFuncVar, rOutput => "HeatingPLC_vAO_Vars".vAO8.rInput)
   END_RUNG
   // the same network as SCL:
   "AOvars"(iFuncSystem := "HeatingPLC_vAO_Vars".vAO8.cFuncSystemID,
            iFuncVar := "HeatingPLC_vAO_Vars".vAO8.cFuncVar,
            rOutput => "HeatingPLC_vAO_Vars".vAO8.rInput);
END_REGION

REGION Network 33
   RUNG wire#powerrail
      "DOvars"(iFuncSystem := "HeatingPLC_vDO_Vars".vDO1.iFuncSystemID, iFuncVar := "HeatingPLC_vDO_Vars".vDO1.iFuncVar, xOutput => "HeatingPLC_vDO_Vars".vDO1.xInput)
   END_RUNG
   // the same network as SCL:
   "DOvars"(iFuncSystem := "HeatingPLC_vDO_Vars".vDO1.iFuncSystemID,
            iFuncVar := "HeatingPLC_vDO_Vars".vDO1.iFuncVar,
            xOutput => "HeatingPLC_vDO_Vars".vDO1.xInput);
END_REGION

REGION Network 34
   RUNG wire#powerrail
      "DOvars"(iFuncSystem := "HeatingPLC_vDO_Vars".vDO2.iFuncSystemID, iFuncVar := "HeatingPLC_vDO_Vars".vDO2.iFuncVar, xOutput => "HeatingPLC_vDO_Vars".vDO2.xInput)
   END_RUNG
   // the same network as SCL:
   "DOvars"(iFuncSystem := "HeatingPLC_vDO_Vars".vDO2.iFuncSystemID,
            iFuncVar := "HeatingPLC_vDO_Vars".vDO2.iFuncVar,
            xOutput => "HeatingPLC_vDO_Vars".vDO2.xInput);
END_REGION

REGION Network 35
   RUNG wire#powerrail
      "DOvars"(iFuncSystem := "HeatingPLC_vDO_Vars".vDO3.iFuncSystemID, iFuncVar := "HeatingPLC_vDO_Vars".vDO3.iFuncVar, xOutput => "HeatingPLC_vDO_Vars".vDO3.xInput)
   END_RUNG
   // the same network as SCL:
   "DOvars"(iFuncSystem := "HeatingPLC_vDO_Vars".vDO3.iFuncSystemID,
            iFuncVar := "HeatingPLC_vDO_Vars".vDO3.iFuncVar,
            xOutput => "HeatingPLC_vDO_Vars".vDO3.xInput);
END_REGION

REGION Network 36
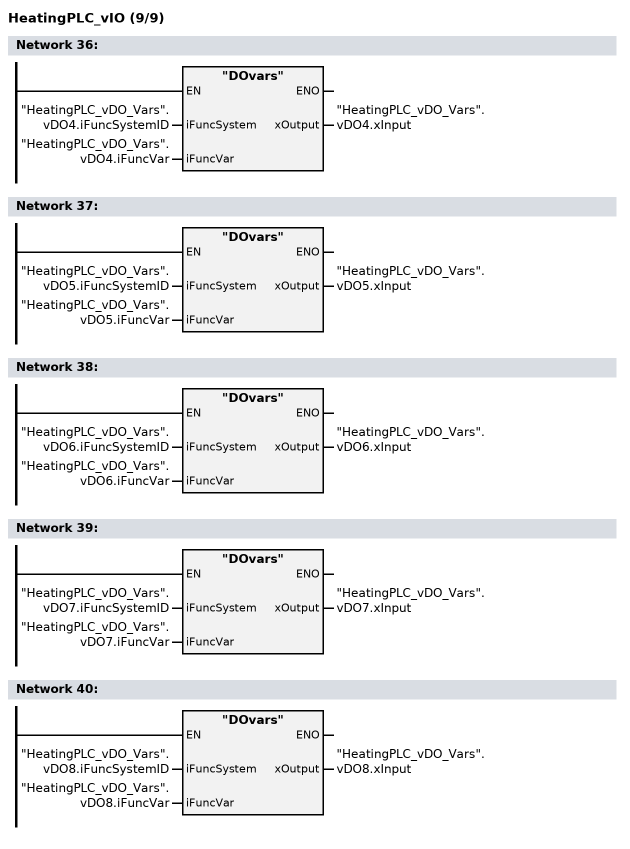
   RUNG wire#powerrail
      "DOvars"(iFuncSystem := "HeatingPLC_vDO_Vars".vDO4.iFuncSystemID, iFuncVar := "HeatingPLC_vDO_Vars".vDO4.iFuncVar, xOutput => "HeatingPLC_vDO_Vars".vDO4.xInput)
   END_RUNG
   // the same network as SCL:
   "DOvars"(iFuncSystem := "HeatingPLC_vDO_Vars".vDO4.iFuncSystemID,
            iFuncVar := "HeatingPLC_vDO_Vars".vDO4.iFuncVar,
            xOutput => "HeatingPLC_vDO_Vars".vDO4.xInput);
END_REGION

REGION Network 37
   RUNG wire#powerrail
      "DOvars"(iFuncSystem := "HeatingPLC_vDO_Vars".vDO5.iFuncSystemID, iFuncVar := "HeatingPLC_vDO_Vars".vDO5.iFuncVar, xOutput => "HeatingPLC_vDO_Vars".vDO5.xInput)
   END_RUNG
   // the same network as SCL:
   "DOvars"(iFuncSystem := "HeatingPLC_vDO_Vars".vDO5.iFuncSystemID,
            iFuncVar := "HeatingPLC_vDO_Vars".vDO5.iFuncVar,
            xOutput => "HeatingPLC_vDO_Vars".vDO5.xInput);
END_REGION

REGION Network 38
   RUNG wire#powerrail
      "DOvars"(iFuncSystem := "HeatingPLC_vDO_Vars".vDO6.iFuncSystemID, iFuncVar := "HeatingPLC_vDO_Vars".vDO6.iFuncVar, xOutput => "HeatingPLC_vDO_Vars".vDO6.xInput)
   END_RUNG
   // the same network as SCL:
   "DOvars"(iFuncSystem := "HeatingPLC_vDO_Vars".vDO6.iFuncSystemID,
            iFuncVar := "HeatingPLC_vDO_Vars".vDO6.iFuncVar,
            xOutput => "HeatingPLC_vDO_Vars".vDO6.xInput);
END_REGION

REGION Network 39
   RUNG wire#powerrail
      "DOvars"(iFuncSystem := "HeatingPLC_vDO_Vars".vDO7.iFuncSystemID, iFuncVar := "HeatingPLC_vDO_Vars".vDO7.iFuncVar, xOutput => "HeatingPLC_vDO_Vars".vDO7.xInput)
   END_RUNG
   // the same network as SCL:
   "DOvars"(iFuncSystem := "HeatingPLC_vDO_Vars".vDO7.iFuncSystemID,
            iFuncVar := "HeatingPLC_vDO_Vars".vDO7.iFuncVar,
            xOutput => "HeatingPLC_vDO_Vars".vDO7.xInput);
END_REGION

REGION Network 40
   RUNG wire#powerrail
      "DOvars"(iFuncSystem := "HeatingPLC_vDO_Vars".vDO8.iFuncSystemID, iFuncVar := "HeatingPLC_vDO_Vars".vDO8.iFuncVar, xOutput => "HeatingPLC_vDO_Vars".vDO8.xInput)
   END_RUNG
   // the same network as SCL:
   "DOvars"(iFuncSystem := "HeatingPLC_vDO_Vars".vDO8.iFuncSystemID,
            iFuncVar := "HeatingPLC_vDO_Vars".vDO8.iFuncVar,
            xOutput => "HeatingPLC_vDO_Vars".vDO8.xInput);
END_REGION
END_FUNCTION
